// LS Electric XG5000 project: 동남100
// PLC NewPLC
// module base 0 slot 0: 입출력 모듈:XBC-DN/DP14E (DC 24V 입력 8점, 트랜지스터 출력 6점)

PROGRAM NewProgram (task: 스캔 프로그램)

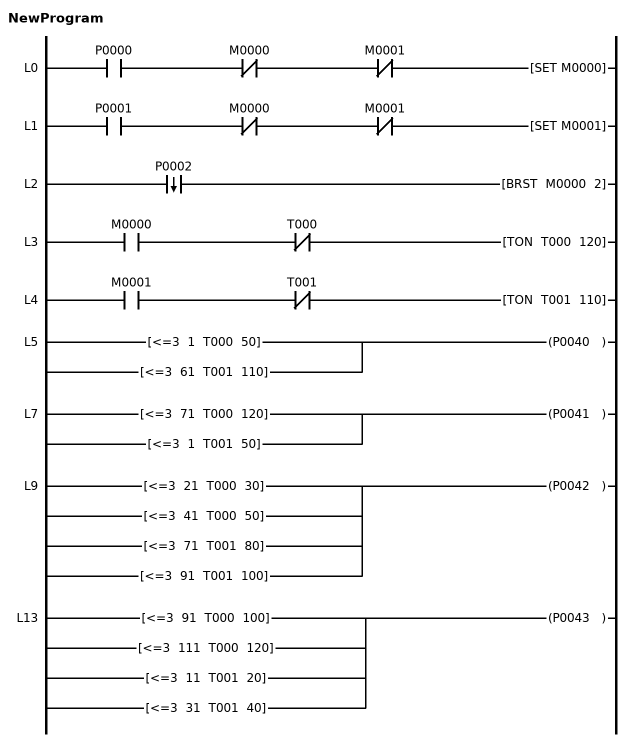
; L0
LOAD      P0000
AND NOT   M0000
AND NOT   M0001
SET       M0000
; L1
LOAD      P0001
AND NOT   M0000
AND NOT   M0001
SET       M0001
; L2
LOADN     P0002
BRST      M0000 2
; L3
LOAD      M0000
AND NOT   T000
TON       T000 120
; L4
LOAD      M0001
AND NOT   T001
TON       T001 110
; L5
LOAD<=3   1 T000 50
OR<=3     61 T001 110
OUT       P0040
; L7
LOAD<=3   71 T000 120
OR<=3     1 T001 50
OUT       P0041
; L9
LOAD<=3   21 T000 30
OR<=3     41 T000 50
OR<=3     71 T001 80
OR<=3     91 T001 100
OUT       P0042
; L13
LOAD<=3   91 T000 100
OR<=3     111 T000 120
OR<=3     11 T001 20
OR<=3     31 T001 40
OUT       P0043